INTERFACE I_Test

END_INTERFACE

(* stored: Version 1.1.0.1, ProductVersion 3.1.4024.11
   Itf I_Test: Id {edea3cf2-efad-4877-b659-e070f43dd056} *)
